PROGRAM HV_Monitor
VAR
	scaled_voltage :INT;
	avg_raw : INT;
	sum_raw : REAL;
	prev_raw : INT;
	i : INT:=0;
END_VAR

//scaled_voltage := REAL_TO_INT(1.6433*raw-12270);
//scaled_voltage := REAL_TO_INT(1.6577*raw-12721);
(*IF (GVL.raw_HV_monitor<=7180 AND GVL.raw_HV_monitor>=7040) THEN
	sum_raw:=0;
	FOR i := 1 TO 20{BY 1)} DO
		sum_raw:= sum_raw+GVL.raw_HV_monitor ;
	END_FOR
	avg_raw:=REAL_TO_INT((sum_raw)/20);
	IF (avg_raw <=7151 AND avg_raw>=7070) THEN
		scaled_voltage:=0; 
	ELSIF (avg_raw <=7116 AND avg_raw>=7052) THEN
		scaled_voltage:=-35;
	ELSIF (avg_raw <=7178 AND avg_raw>=7080) THEN
		scaled_voltage:=35;
	END_IF
ELSE
	scaled_voltage := REAL_TO_INT(0.4748150*GVL.raw_HV_monitor-3558.738574);
END_IF*)
scaled_voltage := REAL_TO_INT(0.4748150*GVL.raw_HV_monitor-3558.738574);

END_PROGRAM

(* stored: Version 1.1.0.1, ProductVersion 3.1.4024.11
   POU HV_Monitor: Id {bda74a86-12a5-4e06-88fc-bf4297d99d5e}, SpecialFunc None *)
